# EPICS substitutions: testDevApp/Db/userHost.substitutions
# Example substitutions file

file "db/dbExample1.db" {
    { user = "lucasHost" }
}

file db/dbExample2.db {
    pattern { user, no, scan }
        { "lucasHost", 1, "1 second" }
        { "lucasHost", 2, "2 second" }
        { "lucasHost", 3, "5 second" }
}
